// TIA Portal V19 export
FUNCTION_BLOCK "TYPIC_C501_IF_HYK"   // FB65, FBD
TITLE = TYPIC_C501_IF_HYK: Hydrantkast tunnelmond
{ S7_Optimized_Access := 'TRUE' }
AUTHOR : OCOTECH
FAMILY : Typical
NAME : C501.709
// Logisch Object Besturing: C501.709
// 
// De interne functie hydrantkast verzorgt de interne bewaking van een hydrantkast.
// stored: MemoryReserve 10, SetENOAutomatically false
   VAR_INPUT
      EXT_HW { ExternalAccessible := 'False'; ExternalVisible := 'False'; ExternalWritable := 'False'} : Bool;   // Sturings hardware (PLC) bewaking (1 = OK)
      IN_DEC { ExternalAccessible := 'False'; ExternalVisible := 'False'; ExternalWritable := 'False'} : Bool;   // De hydrantkast in de verkeerskoker is gesloten. (TRUE = Gesloten)
      IN_STO { ExternalAccessible := 'False'; ExternalVisible := 'False'; ExternalWritable := 'False'} : Bool;   // Temperatuursensor (TRUE = OK / FALSE = Storing)
      IN_AUT_C501 { ExternalAccessible := 'False'; ExternalVisible := 'False'; ExternalWritable := 'False'} : Bool;   // Beveiligingen: serie geschakelde terugmelding (1= OK)
   END_VAR
   VAR_OUTPUT
      VAR_IF_HYK { ExternalAccessible := 'False'; ExternalVisible := 'False'; ExternalWritable := 'False'} : "C501_VAR_IF_HYK_TYPIC";   // Struct met alle variabelen naar bovenliggende functies
   END_VAR
   VAR
      STO { ExternalWritable := 'False'} : Struct   // Storingen
         A001 : Bool;   // Beveiliging aangesproken
         A002 : Bool;   // Temperatuur te laag
      END_STRUCT;
      VAR { ExternalWritable := 'False'} : Struct   // Variabelen
         DEC : Bool;   // De hydrantkast in de verkeerskoker is gesloten
         EXT_HW { ExternalAccessible := 'False'; ExternalVisible := 'False'} : Bool;   // Sturings hardware (PLC) in storing
      END_STRUCT;
   END_VAR
BEGIN

REGION Network 1: START
END_REGION

REGION Network 2: +++ Storingen +++
   // Storingen van de hydrantkast.
END_REGION

REGION Network 3: Storing A001: Beveiliging aangesproken
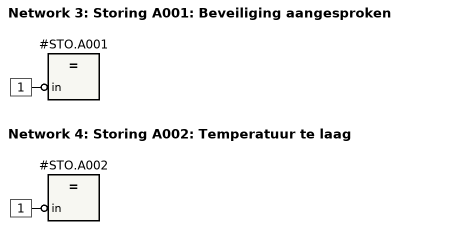
   #STO.A001 := NOT 1;
END_REGION

REGION Network 4: Storing A002: Temperatuur te laag
   #STO.A002 := NOT 1;
END_REGION

REGION Network 5: +++ Variabelen +++
   // Toestandsvariabelen naar 3B sturen
END_REGION

REGION Network 6 (SCL): EINDE
   // Variabelen van intern scada rakvlak naar outputs copieren
   #VAR_IF_HYK.DEC := #VAR.DEC;
   #VAR_IF_HYK.EXT_HW := #VAR.EXT_HW;
   #VAR_IF_HYK.STO := #STO;
END_REGION
END_FUNCTION_BLOCK
